{attribute 'linkalways'}
{attribute 'no_explicit_call' := 'This FB is a CLASS and must be accessed using methods or properties'}
{attribute 'enable_dynamic_creation'}
FUNCTION_BLOCK Node_F_VN_FindReferenceKeyPointsInImageORB EXTENDS VisionNode
VAR
    ipSrcImage : _ITcVnImage;
    ipRefKeyPoints : _ITcVnContainer;
    ipRefDescriptors : _ITcVnImage;
    nRefImageWidth : _UDINT(0);
    nRefImageHeight : _UDINT(0);
    ipEdgePoints : _ITcVnContainer;
    fMaxDist : _REAL(-1.0);
    fMaxKnnRatio : _REAL(-1.0);
    hrPrev : _HRESULT(S_OK);
    aPerspectiveTransform : _TcVnMatrix3x3_LREAL;
    nNumberOfGoodMatches : _UDINT(0);
    nNumberOfInliers : _UDINT(0);
    hresult : _HRESULT(S_OK);
END_VAR

METHOD PUBLIC Clone : I_Node
VAR
    pNode : POINTER TO Node_F_VN_FindReferenceKeyPointsInImageORB;
END_VAR
pNode := __NEW(Node_F_VN_FindReferenceKeyPointsInImageORB);
Clone := pNode^;
END_METHOD

METHOD FB_init : BOOL
VAR_INPUT
    bInitRetains : BOOL;
    bInCopyCode : BOOL;
END_VAR
AddInput('ipSrcImage', ipSrcImage);
AddInput('ipRefKeyPoints', ipRefKeyPoints);
AddInput('ipRefDescriptors', ipRefDescriptors);
AddInput('nRefImageWidth', nRefImageWidth);
AddInput('nRefImageHeight', nRefImageHeight);
AddOutput('ipEdgePoints', ipEdgePoints);
AddParameter('fMaxDist', fMaxDist);
AddParameter('fMaxKnnRatio', fMaxKnnRatio);
AddInput('hrPrev', hrPrev);
AddOutput('aPerspectiveTransform', aPerspectiveTransform);
AddOutput('nNumberOfGoodMatches', nNumberOfGoodMatches);
AddOutput('nNumberOfInliers', nNumberOfInliers);
AddOutput('hresult', hresult);
END_METHOD

METHOD PROTECTED OnExecute
VAR
    perspectiveTransform : TcVnMatrix3x3_LREAL;
    numberOfGoodMatches : UDINT;
    numberOfInliers : UDINT;
END_VAR
hresult.Value := F_VN_FindReferenceKeyPointsInImageORB(
    ipSrcImage := ipSrcImage.Value,
    ipRefKeyPoints := ipRefKeyPoints.Value,
    ipRefDescriptors := ipRefDescriptors.Value,
    nRefImageWidth := nRefImageWidth.Value,
    nRefImageHeight := nRefImageHeight.Value,
    ipEdgePoints := ipEdgePoints.Value,
    fMaxDist := fMaxDist.Value,
    fMaxKnnRatio := fMaxKnnRatio.Value,
    hrPrev := hrPrev.Value,
    aPerspectiveTransform => perspectiveTransform,
    nNumberOfGoodMatches => numberOfGoodMatches,
    nNumberOfInliers => numberOfInliers);

aPerspectiveTransform.Value := perspectiveTransform;
nNumberOfGoodMatches.Value := numberOfGoodMatches;
nNumberOfInliers.Value := numberOfInliers;
END_METHOD

METHOD PUBLIC PreExecutionCheck
VAR_INPUT
    Check : I_PreExecutionChecks;
END_VAR
Check.IsTrue(ipSrcImage.IsValid, 'ipSrcImage must contain an image');
Check.IsTrue(ipSrcImage.HasChannelCount(1), 'ipSrcImage must have 1 channel');
Check.IsTrue(ipRefKeyPoints.IsValid, 'ipRefKeyPoints must contain a container');
Check.IsTrue(ipRefDescriptors.IsValid, 'ipRefDescriptors must contain an image');
Check.IsTrue(nRefImageWidth.Value > 0, 'nRefImageWidth must be greater than 0');
Check.IsTrue(nRefImageHeight.Value > 0, 'nRefImageHeight must be greater than 0');
Check.IsTrue((fMaxDist.Value = -1.0) OR (fMaxDist.Value >= 0.0), 'fMaxDist must be -1 to disable the filter, or at least 0');
Check.IsTrue((fMaxKnnRatio.Value = -1.0) OR
             ((fMaxKnnRatio.Value >= 0.0) AND (fMaxKnnRatio.Value <= 1.0)), 'fMaxKnnRatio must be -1 to disable the filter, or between 0 and 1');
END_METHOD

END_FUNCTION_BLOCK

(* stored: Version 1.1.0.1, ProductVersion 3.1.4026.19
   POU Node_F_VN_FindReferenceKeyPointsInImageORB: Id {958064dc-068b-48f4-8a1e-fcaa4851a21b}, SpecialFunc None
   Folder Constructor: Id {82ea3e11-9dd2-4959-858b-7645271dfeab}
   Method Clone: Id {cf2d06e9-bb99-45aa-8f5c-a556dd881f04}
   Method FB_init: Id {6bb7ac3a-97b8-44d4-adad-bd129a19be59}
   Method OnExecute: Id {e65869cc-0fa0-47e6-8926-2a0e2ead78ef}
   Method PreExecutionCheck: Id {1be7b33b-cb0e-496a-94ee-3f371724040c} *)
